FUNCTION_BLOCK FB_Square EXTENDS FB_Shape

METHOD Draw : STRING
ADSLOGSTR(    msgCtrlMask:=ADSLOG_MSGTYPE_LOG,
              msgFmtStr:='Drawing a %s square',
              strArg:= SUPER^._color.applyColor());
END_METHOD

END_FUNCTION_BLOCK

(* stored: Version 1.1.0.1, ProductVersion 3.1.4024.12
   POU FB_Square: Id {7bc8aa77-dc79-4bf3-94e3-2968c498b2c6}, SpecialFunc None
   Method Draw: Id {bd4f7875-6af9-4c8e-b05c-62abd600c2b5} *)
